(* Logix 5000 project; controller Generic_AOI_V0_1 vendor 1 type 14 code 176 rev 32.11; software revision 32.00; part 8 of 8 *)
(* tags used below, declared in another part *)
   DeviceStatus : DINT;
   IOLReadActive : BOOL;
   IOLWriteActive : BOOL;
   IOL_READ_Request : BOOL;
   IOL_WRITE_Request : BOOL;
   Done : BOOL;
   Error : BOOL;
   Status : DINT;
(* TBEN_Lx_8IOL_AOI, continued *)

ROUTINE Prescan   (* ladder *)
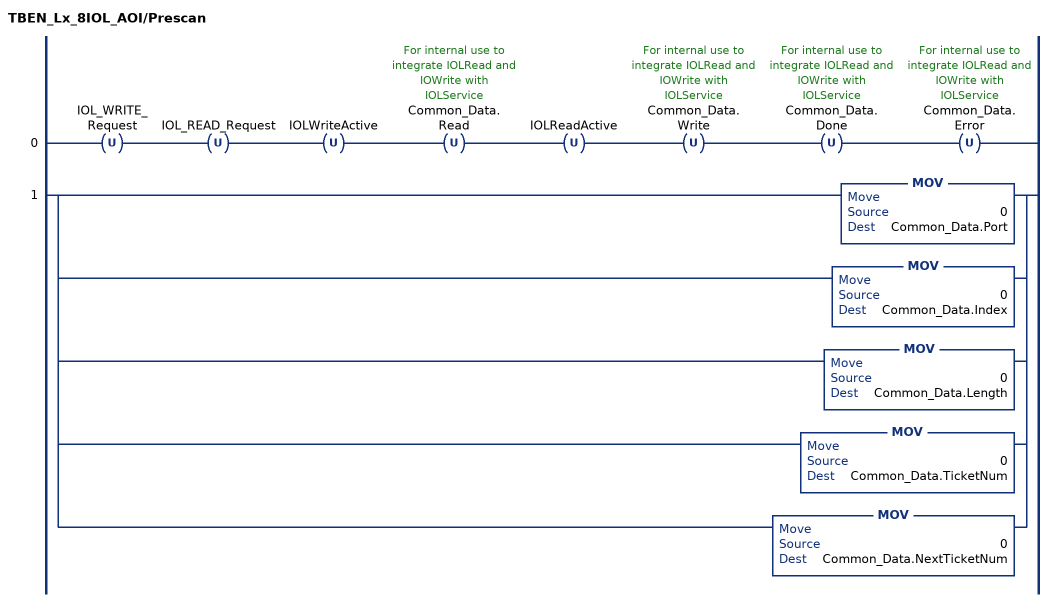
   0: OTU(IOL_WRITE_Request)OTU(IOL_READ_Request)OTU(IOLWriteActive)OTU(Common_Data.Read)OTU(IOLReadActive)OTU(Common_Data.Write)OTU(Common_Data.Done)OTU(Common_Data.Error);
   1: [MOV(0,Common_Data.Port) ,MOV(0,Common_Data.Index) ,MOV(0,Common_Data.Length) ,MOV(0,Common_Data.TicketNum) ,MOV(0,Common_Data.NextTicketNum) ];
END_ROUTINE
END_ADD_ON_INSTRUCTION

ADD_ON_INSTRUCTION Turck_IOL_Generic_AOI   (* revision 1.0 *)
VAR_INPUT
   Port : INT; {required}
END_VAR
VAR_IN_OUT
   Common_Data : Turck_IOLink_Common_Data; {required}
END_VAR
VAR_OUTPUT
   Input_Data_Word0 : INT; {visible}
   Input_Data_Word1 : INT; {visible}
   Input_Data_Word2 : INT; {visible}
   Input_Data_Word3 : INT; {visible}
   Input_Data_Word4 : INT; {visible}
   Input_Data_Word5 : INT; {visible}
   Input_Data_Word6 : INT; {visible}
   Input_Data_Word7 : INT; {visible}
   Input_Data_Word8 : INT;
   Input_Data_Word9 : INT;
   Input_Data_Word10 : INT;
   Input_Data_Word11 : INT;
   Input_Data_Word12 : INT;
   Input_Data_Word13 : INT;
   Input_Data_Word14 : INT;
   Input_Data_Word15 : INT;
END_VAR
VAR_INPUT
   Output_Data_Word0 : INT; {visible}
   Output_Data_Word1 : INT; {visible}
   Output_Data_Word2 : INT; {visible}
   Output_Data_Word3 : INT; {visible}
   Output_Data_Word4 : INT; {visible}
   Output_Data_Word5 : INT; {visible}
   Output_Data_Word6 : INT; {visible}
   Output_Data_Word7 : INT; {visible}
   Output_Data_Word8 : INT;
   Output_Data_Word9 : INT;
   Output_Data_Word10 : INT;
   Output_Data_Word11 : INT;
   Output_Data_Word12 : INT;
   Output_Data_Word13 : INT;
   Output_Data_Word14 : INT;
   Output_Data_Word15 : INT;
   Swap_16 : BOOL; {visible}
   Swap_32 : BOOL; {visible}
   Swap_All : BOOL; {visible}
   Direct : BOOL; {visible}
END_VAR
VAR
   Port_Less_One : INT; {access None}
   Port_Bit : SINT; {access None}
END_VAR

ROUTINE Logic   (* ladder *)
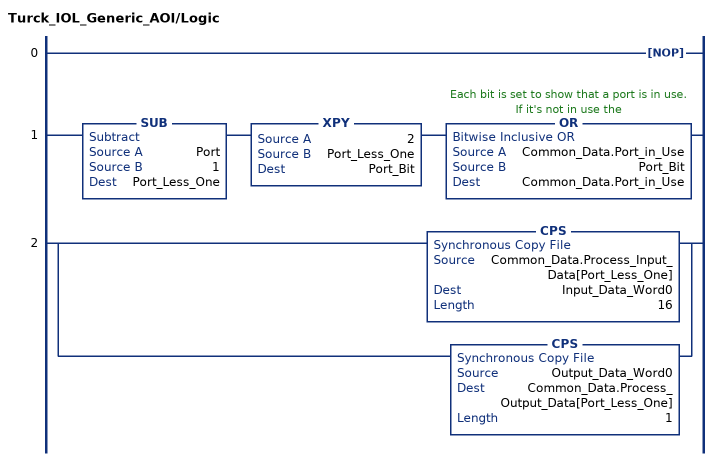
   0: NOP();
   1: SUB(Port,1,Port_Less_One)XPY(2,Port_Less_One,Port_Bit)OR(Common_Data.Port_in_Use,Port_Bit,Common_Data.Port_in_Use);
   2: [CPS(Common_Data.Process_Input_Data[Port_Less_One],Input_Data_Word0,16) ,CPS(Output_Data_Word0,Common_Data.Process_Output_Data[Port_Less_One],1) ];
END_ROUTINE
END_ADD_ON_INSTRUCTION

VAR_GLOBAL   (* controller tags *)
   Common_Data : Turck_IOLink_Common_Data := (Read := 1, Port_in_Use := 1, Port := 128, Index := -1, SubIndex := 68, Status := 1000, NextTicketNum := 1, SendData[0] := -1, SendData[1] := -1, SendData[2] := 68);
   IOL_READ_MSG : MESSAGE;
        MessageParameters(ServiceCode := 16#004b, LocalElement := Common_Data.SendData, DestinationTag := Common_Data.ReceiveData, ...)
   IOL_WRITE_MSG : MESSAGE;
        MessageParameters(ServiceCode := 16#004c, LocalElement := Common_Data.SendData, DestinationTag := Common_Data.ReceiveData, ...)
   Port1_Device : Turck_IOL_Generic_AOI := (Port := 1);
   TBEN_100_8IOL_AOI : TBEN_Lx_8IOL_AOI := (DeviceStatus := 16384);
END_VAR

PROGRAM MainProgram   (* main routine MainRoutine *)

ROUTINE MainRoutine   (* ladder *)
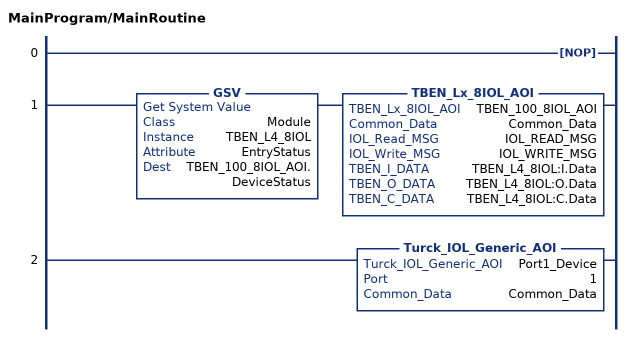
   0: NOP();
   1: GSV(Module,TBEN_L4_8IOL,EntryStatus,TBEN_100_8IOL_AOI.DeviceStatus)TBEN_Lx_8IOL_AOI(TBEN_100_8IOL_AOI,Common_Data,IOL_READ_MSG,IOL_WRITE_MSG,TBEN_L4_8IOL:I.Data,TBEN_L4_8IOL:O.Data,TBEN_L4_8IOL:C.Data);
   2: Turck_IOL_Generic_AOI(Port1_Device,1,Common_Data);
END_ROUTINE
END_PROGRAM

PROGRAM SafetyProgram   (* main routine MainRoutine, safety *)

ROUTINE MainRoutine   (* ladder *)
END_ROUTINE
END_PROGRAM
